{attribute 'linkalways'} 
{attribute 'no_explicit_call' := 'This FB is a CLASS and must be accessed using methods or properties'}
{attribute 'enable_dynamic_creation'}
FUNCTION_BLOCK NullError EXTENDS Error
VAR
END_VAR

PROPERTY ErrorType : T_MAXSTRING
GET
END_GET
END_PROPERTY

PROPERTY PUBLIC Message : T_MAXSTRING
GET
END_GET
END_PROPERTY

METHOD PUBLIC SerializeWith
VAR_INPUT
	Serializer : I_Serializer;
END_VAR
END_METHOD

END_FUNCTION_BLOCK

(* stored: Version 1.1.0.1, ProductVersion 3.1.4024.12
   POU NullError: Id {f1eb6478-889c-09b3-2285-65723a449f23}, SpecialFunc None
   Property ErrorType: Id {cf2a3040-2b0d-04d6-00b5-5d6f9d668c8d}
   Get Get: Id {9ede09e7-92c0-02ab-35ad-10065e0984b9}
   Property Message: Id {752ab385-19e2-0867-2470-f6b2cde8f377}
   Get Get: Id {16b9f71f-dcef-0483-04ed-a5dee0fb501b}
   Method SerializeWith: Id {2d0a2fc1-296a-035d-194d-1de2c0a2f08c} *)
